KUKA KRL program: XmlDualMove_better.src

&ACCESS RV
&REL 1
&PARAM DISKPATH = KRC:\R1\Program
&PARAM SensorITMASK = *
&PARAM TEMPLATE = C:\KRC\Roboter\Template\vorgabe
DEF XmlDualMove_better( )

; ============================================================================
; XmlDualMove_better - robot-interpreter side of the ROS2 link, BATCH capable
; ============================================================================
; RELATIONSHIP WITH XmlDualMove.src
;   XmlDualMove.src        baseline used for the KRL vs MoveIt2 comparative
;                          study.  Untouched.  Still selectable and still
;                          works against XmlDualMove_better.xml, because that
;                          channel config is a strict superset.
;   XmlDualMove_better.src this file: everything the baseline does, PLUS the
;                          batch mode.  Only ONE of the two is selected at a
;                          time; they never run together.
;
; WHAT BATCH MODE CHANGES
;   The baseline executes one point per network round trip: ROS sends a point,
;   waits for the robot to arrive, then sends the next.  Over 100+ trajectory
;   points that dead time is what produces the advance-brake-advance pattern.
;
;   In batch mode ROS ships a block of up to XD_BATCH_MAX points, the SPS drops
;   the whole block into the mailbox in one go, and this program walks it
;   locally with no network in the inner loop.
;
;   Every point is STILL an exact-stop PTP.  No C_PTP, no blending, no SLIN,
;   no Cartesian.  The motion type is identical; only the waiting changes.
;
; ADVANCE RUN
;   KRL executes assignments during the advance run, and $ADVANCE defaults to
;   3 (KSS 8.2 System Integrators, 7.5.3 "Advance run", p. 208: default 3,
;   maximum 5).  Left alone, XD_BATCH_CONSUMED_COUNT would run up to $ADVANCE
;   points ahead of the real motion and the abort check would read stale state.
;
;   This program does NOT write $ADVANCE.  It forces the advance-run stop once
;   per point with WAIT SEC 0 instead, which is the documented way to make an
;   instruction run in the main run, and which costs nothing here because every
;   point is already an exact stop.  $ADVANCE = 0 would be legal (0 is inside
;   the documented range) but it also makes approximate positioning impossible,
;   and blending is where this design is headed next.
;
;   The WAIT SEC 0.1 of the main loop is NOT touched: same place, same value.
;   It simply does not sit between the points of one batch.
; ============================================================================
; THIS PROGRAM CONTAINS NO EthernetKRL CALLS.
;
; SPS.SUB owns the EKI channel: it opens it, drains the receive buffer on
; every cycle and publishes the last valid command into the XD_ mailbox in
; $CONFIG.DAT.  This program only reads that mailbox.  Consequences:
;
;   * Telemetry no longer depends on this program running.  DEMO26 or any
;     other KRL program can be selected and Ubuntu keeps receiving data.
;   * The receive buffer is never blocked by the robot interpreter, which is
;     what used to fill the EKI memory and raise EKI01280.
;   * The manual warns against reading one channel from both interpreters
;     (EKI_Get empties the memory), so all reading stays in the SPS.
;
; SAFETY MODEL
;   * On start-up the current mailbox Seq is taken as a BASELINE and is never
;     executed.  A command that arrived while DEMO26 was running can never
;     move the robot just because this program was selected afterwards.
;   * A Seq is marked handled BEFORE acting on it, so a given Seq can move
;     the robot or drive the gripper at most once.  The Ubuntu heartbeat
;     deliberately repeats the same Seq and is therefore inert.
;   * Gripper and motion are independent: EnableMove=FALSE with
;     GripperCommand 0 or 1 performs a gripper-only action.
;
; ORDER OF EXECUTION for a new Seq:  validate -> gripper -> motion.
; ============================================================================

;FOLD Declaration
  INT i
  INT cmdSeq
  INT cmdSeqCheck
  INT handledSeq
  INT gripperCmd

  DECL AXIS axisTarget
  DECL E6POS cartesianTarget

  BOOL snapshotOK
  BOOL isAxisMode
  BOOL isCartesianMode

  BOOL enableMove
  BOOL limitsOK
  BOOL readyToMove
  BOOL moveExecuted
  BOOL deltaOK
  BOOL velocityOK
  BOOL hasTrajectoryVelocity

  REAL targetA1
  REAL targetA2
  REAL targetA3
  REAL targetA4
  REAL targetA5
  REAL targetA6

  REAL targetX
  REAL targetY
  REAL targetZ
  REAL targetA
  REAL targetB
  REAL targetC
  REAL ptpVelocityPct

  REAL errorA1
  REAL errorA2
  REAL errorA3
  REAL errorA4
  REAL errorA5
  REAL errorA6

  REAL errorX
  REAL errorY
  REAL errorZ
  REAL errorA
  REAL errorB
  REAL errorC

  REAL MAX_DELTA_JOINT
  REAL MAX_DELTA_POS
  REAL MAX_DELTA_ORI

  ; ---- BATCH MODE ----
  INT batchSeq
  INT batchSeqCheck
  INT handledBatchSeq
  INT batchCount
  INT batchI
  INT savedAdvance
  REAL batchVelPct
  REAL batchErr
  BOOL batchSnapshotOK
  BOOL batchRunning
  BOOL batchPointOK
  BOOL hasBatchVelocity
  BOOL batchLoaded
  BOOL batchGateOK
  BOOL batchVelocityOK
  ; Ultimo punto ENTREGADO al planificador.  La validacion de salto se hace
  ; contra este valor y NO contra $AXIS_ACT: con aproximacion activa el robot
  ; va por detras del interprete a proposito, asi que $AXIS_ACT no dice donde
  ; estara cuando se ejecute el punto que se esta validando.  Ademas leer
  ; $AXIS_ACT dentro del encadenado obligaria a una parada del avance, que es
  ; justo lo que impide aproximar (KSS 8.2 SI, 8.5, p. 224).
  REAL prevA1
  REAL prevA2
  REAL prevA3
  REAL prevA4
  REAL prevA5
  REAL prevA6
  INT localBatchSeq
  INT localBatchCount
  REAL localBatchVelPct
  DECL AXIS batchTarget

  ; LOCAL copy of the batch.  The mailbox holds ONE batch slot, so executing
  ; straight out of it would mean ROS could not load the next batch until the
  ; current one finished - the very network gap batch mode exists to remove.
  ; Copying to locals frees the mailbox the moment execution starts, so ROS
  ; can refill it while the robot is still moving.
  REAL localA1[20]
  REAL localA2[20]
  REAL localA3[20]
  REAL localA4[20]
  REAL localA5[20]
  REAL localA6[20]
;ENDFOLD (Declaration)

;FOLD INI
  ;FOLD BASISTECH INI
    BAS (#INITMOV,0 )
  ;ENDFOLD (BASISTECH INI)

  ;FOLD USER INI
    ;Reads targets from the XD_ mailbox published by SPS.SUB.
    ;Supports BOTH Axis (A1-A6) and Cartesian (X,Y,Z,A,B,C) modes.
    ;Movement must be enabled by the responsible operator via the bridge.
  ;ENDFOLD (USER INI)
;ENDFOLD (INI)

;FOLD Initialize data
  cmdSeq = 0
  cmdSeqCheck = 0
  gripperCmd = -1

  snapshotOK = FALSE
  enableMove = FALSE
  limitsOK = FALSE
  readyToMove = FALSE
  moveExecuted = FALSE
  deltaOK = FALSE
  velocityOK = FALSE
  hasTrajectoryVelocity = FALSE
  isAxisMode = FALSE
  isCartesianMode = FALSE

  targetA1 = $AXIS_ACT.A1
  targetA2 = $AXIS_ACT.A2
  targetA3 = $AXIS_ACT.A3
  targetA4 = $AXIS_ACT.A4
  targetA5 = $AXIS_ACT.A5
  targetA6 = $AXIS_ACT.A6

  targetX = $POS_ACT.X
  targetY = $POS_ACT.Y
  targetZ = $POS_ACT.Z
  targetA = $POS_ACT.A
  targetB = $POS_ACT.B
  targetC = $POS_ACT.C
  ptpVelocityPct = 0.0

  errorA1 = 0.0
  errorA2 = 0.0
  errorA3 = 0.0
  errorA4 = 0.0
  errorA5 = 0.0
  errorA6 = 0.0

  errorX = 0.0
  errorY = 0.0
  errorZ = 0.0
  errorA = 0.0
  errorB = 0.0
  errorC = 0.0

  MAX_DELTA_JOINT = 10.0
  MAX_DELTA_POS = 100.0  ; 100 mm jump max in X, Y, Z
  MAX_DELTA_ORI = 20.0   ; 20 degrees jump max in A, B, C

  axisTarget = $AXIS_ACT
  cartesianTarget = $POS_ACT

  ; ---- BASELINE ----
  ; Whatever is sitting in the mailbox right now belongs to the past: it may
  ; have arrived while DEMO26 was running, or be the last command of an
  ; earlier ROS2 session.  Treating it as already handled is what stops this
  ; program from moving the moment it is selected.
  handledSeq = XD_CMD_SEQ

  ; Same baseline rule for the batch: whatever batch is sitting in the mailbox
  ; when this program is selected belongs to the past and is never executed.
  handledBatchSeq = XD_BATCH_SEQ

  batchSeq = 0
  batchSeqCheck = 0
  batchCount = 0
  batchI = 0
  savedAdvance = 3
  batchVelPct = 0.0
  batchErr = 0.0
  batchSnapshotOK = FALSE
  batchRunning = FALSE
  batchPointOK = FALSE
  hasBatchVelocity = FALSE
  batchLoaded = FALSE
  batchGateOK = FALSE
  batchVelocityOK = FALSE
  prevA1 = 0.0
  prevA2 = 0.0
  prevA3 = 0.0
  prevA4 = 0.0
  prevA5 = 0.0
  prevA6 = 0.0
  localBatchSeq = 0
  localBatchCount = 0
  localBatchVelPct = 0.0
  batchTarget = $AXIS_ACT

  XD_BATCH_ACTIVE = FALSE
  XD_BATCH_CONSUMED_COUNT = 0

  XD_MOVE_READY = FALSE
  XD_LIMITS_OK = FALSE
  XD_DELTA_OK = FALSE
;ENDFOLD (Initialize data)

;FOLD Configure motion parameters
  $BWDSTART = FALSE

  ; Default TOOL and BASE (modify if your setup requires specific ones)
  $TOOL = $NULLFRAME
  $BASE = $NULLFRAME
;ENDFOLD (Configure motion parameters)

;FOLD Move command loop
LOOP

  ;FOLD Snapshot the mailbox
    ; Seqlock read: XD_CMD_SEQ is written LAST by the SPS, so reading it
    ; before and after the payload detects a publish that landed mid-copy.
    ; A torn snapshot is simply discarded and retried next cycle.
    snapshotOK = FALSE

    IF XD_CMD_UPDATING == FALSE THEN
      cmdSeqCheck = XD_CMD_SEQ

      targetA1 = XD_TARGET_A1
      targetA2 = XD_TARGET_A2
      targetA3 = XD_TARGET_A3
      targetA4 = XD_TARGET_A4
      targetA5 = XD_TARGET_A5
      targetA6 = XD_TARGET_A6

      targetX = XD_TARGET_X
      targetY = XD_TARGET_Y
      targetZ = XD_TARGET_Z
      targetA = XD_TARGET_A
      targetB = XD_TARGET_B
      targetC = XD_TARGET_C

      enableMove = XD_ENABLE_MOVE
      gripperCmd = XD_GRIPPER_COMMAND
      ptpVelocityPct = XD_TRAJ_PTP_VEL_PCT
      isAxisMode = XD_AXIS_MODE
      isCartesianMode = XD_CART_MODE

      IF (XD_CMD_UPDATING == FALSE) AND (XD_CMD_SEQ == cmdSeqCheck) THEN
        cmdSeq = cmdSeqCheck
        snapshotOK = TRUE
      ENDIF
    ENDIF
  ;ENDFOLD (Snapshot the mailbox)

  ;FOLD Snapshot the batch mailbox
    ; Same seqlock idea as the single-point snapshot: XD_BATCH_SEQ is written
    ; LAST by the SPS, so reading it before and after the payload detects a
    ; publish that landed mid-copy.  A torn batch is discarded and retried.
    batchSnapshotOK = FALSE

    IF XD_CMD_UPDATING == FALSE THEN
      batchSeqCheck = XD_BATCH_SEQ
      batchCount = XD_BATCH_COUNT
      batchVelPct = XD_BATCH_PTP_VEL_PCT

      IF (XD_CMD_UPDATING == FALSE) AND (XD_BATCH_SEQ == batchSeqCheck) THEN
        batchSeq = batchSeqCheck
        batchSnapshotOK = TRUE
      ENDIF
    ENDIF

    ; A batch mailbox reset follows the same rule as the single-point one.
    IF batchSnapshotOK == TRUE THEN
      IF batchSeq == 0 THEN
        handledBatchSeq = 0
      ENDIF
    ENDIF

    ; Velocity validation, identical rule to the single-point path.
    hasBatchVelocity = FALSE
    IF (batchVelPct > 0.0) AND (batchVelPct <= 100.0) THEN
      hasBatchVelocity = TRUE
    ENDIF
  ;ENDFOLD (Snapshot the batch mailbox)

  ;FOLD Follow a mailbox reset
    ; XD_CMD_SEQ == 0 is the sentinel the SPS writes when it (re)opens the
    ; channel: the mailbox holds no command at all.  There is nothing from
    ; the past to protect against, so the handled marker follows it down.
    ; Without this, a fresh ROS2 session that restarts its counter at 1 could
    ; have its very first command silently ignored.
    IF snapshotOK == TRUE THEN
      IF cmdSeq == 0 THEN
        handledSeq = 0
      ENDIF
    ENDIF
  ;ENDFOLD (Follow a mailbox reset)

  ;FOLD Calculate error target - actual
    IF isAxisMode THEN
      errorA1 = targetA1 - $AXIS_ACT.A1
      errorA2 = targetA2 - $AXIS_ACT.A2
      errorA3 = targetA3 - $AXIS_ACT.A3
      errorA4 = targetA4 - $AXIS_ACT.A4
      errorA5 = targetA5 - $AXIS_ACT.A5
      errorA6 = targetA6 - $AXIS_ACT.A6
    ENDIF

    IF isCartesianMode THEN
      errorX = targetX - $POS_ACT.X
      errorY = targetY - $POS_ACT.Y
      errorZ = targetZ - $POS_ACT.Z
      errorA = targetA - $POS_ACT.A
      errorB = targetB - $POS_ACT.B
      errorC = targetC - $POS_ACT.C
    ENDIF
  ;ENDFOLD (Calculate error target - actual)

  ;FOLD Validate limits
    limitsOK = TRUE

    IF isAxisMode THEN
      IF targetA1 < -160.0 THEN
        limitsOK = FALSE
      ENDIF
      IF targetA1 > 160.0 THEN
        limitsOK = FALSE
      ENDIF
      IF targetA2 < -180.0 THEN
        limitsOK = FALSE
      ENDIF
      IF targetA2 > 35.0 THEN
        limitsOK = FALSE
      ENDIF
      IF targetA3 < -110.0 THEN
        limitsOK = FALSE
      ENDIF
      IF targetA3 > 146.0 THEN
        limitsOK = FALSE
      ENDIF
      IF targetA4 < -175.0 THEN
        limitsOK = FALSE
      ENDIF
      IF targetA4 > 175.0 THEN
        limitsOK = FALSE
      ENDIF
      IF targetA5 < -110.0 THEN
        limitsOK = FALSE
      ENDIF
      IF targetA5 > 110.0 THEN
        limitsOK = FALSE
      ENDIF
      IF targetA6 < -340.0 THEN
        limitsOK = FALSE
      ENDIF
      IF targetA6 > 340.0 THEN
        limitsOK = FALSE
      ENDIF
    ENDIF

    ; Note: Cartesian limits are harder to define safely without a known workspace.
    ; Native KUKA reachability will prevent unsafe poses, but you can add boundary boxes here if needed.
  ;ENDFOLD (Validate limits)

  XD_LIMITS_OK = limitsOK

  ;FOLD Validate delta (max jump per command)
    deltaOK = TRUE

    IF isAxisMode THEN
      IF (errorA1 > MAX_DELTA_JOINT) OR (errorA1 < -MAX_DELTA_JOINT) THEN
        deltaOK = FALSE
      ENDIF
      IF (errorA2 > MAX_DELTA_JOINT) OR (errorA2 < -MAX_DELTA_JOINT) THEN
        deltaOK = FALSE
      ENDIF
      IF (errorA3 > MAX_DELTA_JOINT) OR (errorA3 < -MAX_DELTA_JOINT) THEN
        deltaOK = FALSE
      ENDIF
      IF (errorA4 > MAX_DELTA_JOINT) OR (errorA4 < -MAX_DELTA_JOINT) THEN
        deltaOK = FALSE
      ENDIF
      IF (errorA5 > MAX_DELTA_JOINT) OR (errorA5 < -MAX_DELTA_JOINT) THEN
        deltaOK = FALSE
      ENDIF
      IF (errorA6 > MAX_DELTA_JOINT) OR (errorA6 < -MAX_DELTA_JOINT) THEN
        deltaOK = FALSE
      ENDIF
    ENDIF

    IF isCartesianMode THEN
      IF (errorX > MAX_DELTA_POS) OR (errorX < -MAX_DELTA_POS) THEN
        deltaOK = FALSE
      ENDIF
      IF (errorY > MAX_DELTA_POS) OR (errorY < -MAX_DELTA_POS) THEN
        deltaOK = FALSE
      ENDIF
      IF (errorZ > MAX_DELTA_POS) OR (errorZ < -MAX_DELTA_POS) THEN
        deltaOK = FALSE
      ENDIF
      IF (errorA > MAX_DELTA_ORI) OR (errorA < -MAX_DELTA_ORI) THEN
        deltaOK = FALSE
      ENDIF
      IF (errorB > MAX_DELTA_ORI) OR (errorB < -MAX_DELTA_ORI) THEN
        deltaOK = FALSE
      ENDIF
      IF (errorC > MAX_DELTA_ORI) OR (errorC < -MAX_DELTA_ORI) THEN
        deltaOK = FALSE
      ENDIF
    ENDIF
  ;ENDFOLD (Validate delta)

  XD_DELTA_OK = deltaOK

  ;FOLD Validate trajectory PTP velocity
    ; 0.0 identifies SEND manual/legacy and leaves the current programmed PTP
    ; velocity untouched. Positive values belong only to AxisTarget trajectory
    ; commands. Invalid mailbox values block motion.
    velocityOK = FALSE
    hasTrajectoryVelocity = FALSE

    IF ptpVelocityPct == 0.0 THEN
      velocityOK = TRUE
    ENDIF
    IF (ptpVelocityPct > 0.0) AND (ptpVelocityPct <= 100.0) THEN
      velocityOK = TRUE
      hasTrajectoryVelocity = TRUE
    ENDIF
    IF isCartesianMode AND hasTrajectoryVelocity THEN
      velocityOK = FALSE
    ENDIF
  ;ENDFOLD (Validate trajectory PTP velocity)

  ;FOLD Build target from mailbox
    IF isAxisMode THEN
      axisTarget = $AXIS_ACT
      axisTarget.A1 = targetA1
      axisTarget.A2 = targetA2
      axisTarget.A3 = targetA3
      axisTarget.A4 = targetA4
      axisTarget.A5 = targetA5
      axisTarget.A6 = targetA6
    ENDIF

    IF isCartesianMode THEN
      cartesianTarget = $POS_ACT
      cartesianTarget.X = targetX
      cartesianTarget.Y = targetY
      cartesianTarget.Z = targetZ
      cartesianTarget.A = targetA
      cartesianTarget.B = targetB
      cartesianTarget.C = targetC
    ENDIF
  ;ENDFOLD (Build target from mailbox)

  ;FOLD Determine readyToMove
    readyToMove = FALSE

    IF enableMove == TRUE THEN
      IF limitsOK == TRUE THEN
        IF deltaOK == TRUE THEN
          IF velocityOK == TRUE THEN
            IF snapshotOK == TRUE THEN
              readyToMove = TRUE
            ENDIF
          ENDIF
        ENDIF
      ENDIF
    ENDIF

    IF XD_EKI_ACTIVE == FALSE THEN
      readyToMove = FALSE
    ENDIF
    IF (isAxisMode == FALSE) AND (isCartesianMode == FALSE) THEN
      readyToMove = FALSE
    ENDIF

    XD_MOVE_READY = readyToMove
  ;ENDFOLD (Determine readyToMove)

  ;FOLD Act on a NEW sequence only
    ; A Seq is acted on exactly once.  handledSeq is advanced BEFORE the
    ; action, so nothing can replay it: not the heartbeat, not a restart.
    ;
    ; BATCH GUARD: a batch packet also carries Command/Seq, so without this
    ; guard the single-point block would fire on the batch packet and drive
    ; the robot to XD_TARGET_A1..A6 before the batch even starts.  While a
    ; batch is pending or running, the single-point path stands down.
    ; Ordinary single-point commands are unaffected: with no batch in the
    ; mailbox, batchSeq equals handledBatchSeq and this guard is transparent.
    IF (batchSeq == handledBatchSeq) AND (batchRunning == FALSE) THEN
    IF snapshotOK == TRUE THEN
      IF cmdSeq > 0 THEN
        IF cmdSeq <> handledSeq THEN
          IF XD_EKI_ACTIVE == TRUE THEN

            handledSeq = cmdSeq

            ;FOLD Gripper action
              ; -1 = do nothing (the bridge default), 0 = open, 1 = close.
              ; The SPS has already rejected any other value.
              IF gripperCmd == 0 THEN
                GRPg_SetStateAndCheck(1, 1, 0.2, 1)
              ENDIF
              IF gripperCmd == 1 THEN
                GRPg_SetStateAndCheck(1, 2, 0.2, 1)
              ENDIF
            ;ENDFOLD (Gripper action)

            ;FOLD Motion
              IF readyToMove == TRUE THEN
                IF isAxisMode THEN
                  IF hasTrajectoryVelocity THEN
                    BAS (#VEL_PTP,ptpVelocityPct)
                  ENDIF
                  PTP axisTarget
                ENDIF

                IF isCartesianMode THEN
                  PTP cartesianTarget
                ENDIF

                moveExecuted = TRUE
                XD_LAST_MOVE_SEQ = cmdSeq
                XD_MOVE_EXECUTED = TRUE
              ENDIF
            ;ENDFOLD (Motion)

          ENDIF
        ENDIF
      ENDIF
    ENDIF
    ENDIF
  ;ENDFOLD (Act on a NEW sequence only)

  ;FOLD Execute a NEW batch
    ; A batch is acted on exactly once, same contract as a single Seq:
    ; handledBatchSeq advances BEFORE the first point, so nothing can replay
    ; it after a restart or a repeated packet.
    ;
    ; REFILL WHILE MOVING
    ;   The mailbox has ONE batch slot.  Executing straight out of it would
    ;   force ROS to wait for the batch to finish before loading the next,
    ;   reintroducing one network gap per batch.  So the batch is copied into
    ;   local arrays first: the mailbox is free again immediately and ROS can
    ;   refill it while the robot is still moving through the local copy.
    ;   The WHILE below then picks up that next batch with no gap at all.
    ;
    ;   If no new batch has arrived by the time the local copy runs out, the
    ;   WHILE exits and the outer loop simply waits - same behaviour as the
    ;   baseline when no command is present.
    ; Entry gate for a new batch.  These five conditions were five nested
    ; IFs.  KRL allows at most 10 nested control structures and that pushed
    ; the batch loop to depth 12, so the controller rejected the file with
    ; error 2218.  Same conditions, same order, same outcome - the only
    ; thing that changed is the nesting depth.  Do NOT re-nest them.
    batchGateOK = (batchSnapshotOK == TRUE) AND (batchSeq > 0)
    batchGateOK = batchGateOK AND (batchSeq <> handledBatchSeq)
    batchGateOK = batchGateOK AND (XD_EKI_ACTIVE == TRUE)
    batchGateOK = batchGateOK AND (XD_ENABLE_MOVE == TRUE)
    IF batchGateOK == TRUE THEN

      ; EL LOTE CONSUME TAMBIEN Command/Seq.
      ; Un paquete de lote lleva ADEMAS Command/Seq y Command/AxisTarget.
      ; Ese AxisTarget es relleno inerte: la posicion que tenia el robot
      ; cuando ROS envio el lote.  Pero el bloque de punto suelto no sabe
      ; que es relleno.  Al terminar el lote su puerta se reabre
      ; (batchSeq == handledBatchSeq, batchRunning == FALSE), encuentra un
      ; Seq que nadie ha atendido y lo ejecuta como un PTP normal: el robot
      ; vuelve al punto donde EMPEZO el lote.
      ; En los tramos largos la validacion de delta lo frena (recorridos de
      ; 30-90 grados contra MAX_DELTA_JOINT = 10.0).  En los tramos cortos
      ; de aproximacion y retirada NO: P3->P4 son 9.888 grados, y P4->P5
      ; otros 9.710.  Medido: el robot bajaba, agarraba, subia, volvia a
      ; bajar y a subir varias veces antes de seguir - un rebote por cada
      ; tramo corto.
      ; Atender el Seq aqui es correcto por definicion: el paquete YA se ha
      ; consumido, por el camino de lote.  Nada se pierde, porque el
      ; AxisTarget de un paquete de lote nunca fue un destino real y su
      ; GripperCommand es siempre -1.
      handledSeq = cmdSeq

      ; A stale abort from a previous batch must not kill this one.
      XD_ABORT_BATCH = FALSE
      XD_BATCH_ACTIVE = TRUE
      batchRunning = TRUE

      ; Every point inside the batch forces its own advance-run stop
      ; with WAIT SEC 0 (see the FOR below).  $ADVANCE is deliberately
      ; NOT written here.  It was once suspected of raising KSS01422;
      ; that was never proven - the error kept firing after every write
      ; to $ADVANCE had been removed - so that claim is withdrawn.
      ; WAIT SEC 0 stays because it is the documented mechanism, not
      ; because $ADVANCE is dangerous.

      ; Ancla de la cadena de validacion.  Esta es la UNICA lectura de
      ; $AXIS_ACT de todo el camino de movimiento, y esta antes del primer
      ; PTP, donde una parada del avance no cuesta nada.  A partir de aqui
      ; cada punto se valida contra el ANTERIOR, que es exactamente lo que
      ; preflight() de ROS ya comprueba sobre el archivo entero.
      WAIT SEC 0
      prevA1 = $AXIS_ACT.A1
      prevA2 = $AXIS_ACT.A2
      prevA3 = $AXIS_ACT.A3
      prevA4 = $AXIS_ACT.A4
      prevA5 = $AXIS_ACT.A5
      prevA6 = $AXIS_ACT.A6

      WHILE batchRunning == TRUE

        ;FOLD Copy the mailbox batch into the local arrays
          ; Seqlock read, same idea as the single-point snapshot.
          batchLoaded = FALSE

          IF XD_CMD_UPDATING == FALSE THEN
            batchSeqCheck = XD_BATCH_SEQ
            localBatchCount = XD_BATCH_COUNT
            localBatchVelPct = XD_BATCH_PTP_VEL_PCT

            IF localBatchCount > 0 THEN
              IF localBatchCount <= XD_BATCH_MAX THEN
                FOR batchI = 1 TO localBatchCount
                  localA1[batchI] = XD_BATCH_A1[batchI]
                  localA2[batchI] = XD_BATCH_A2[batchI]
                  localA3[batchI] = XD_BATCH_A3[batchI]
                  localA4[batchI] = XD_BATCH_A4[batchI]
                  localA5[batchI] = XD_BATCH_A5[batchI]
                  localA6[batchI] = XD_BATCH_A6[batchI]
                ENDFOR

                IF (XD_CMD_UPDATING == FALSE) AND (XD_BATCH_SEQ == batchSeqCheck) THEN
                  IF batchSeqCheck <> handledBatchSeq THEN
                    localBatchSeq = batchSeqCheck
                    batchLoaded = TRUE
                  ENDIF
                ENDIF
              ENDIF
            ENDIF
          ENDIF

          ; Nothing new in the mailbox: leave the batch loop and let
          ; the outer loop wait.  The robot does not move.
          IF batchLoaded == FALSE THEN
            batchRunning = FALSE
          ENDIF
        ;ENDFOLD (Copy the mailbox batch)

        IF batchRunning == TRUE THEN

          ; Claimed BEFORE the first point: nothing can replay it.
          handledBatchSeq = localBatchSeq

          ; XD_BATCH_CONSUMED_COUNT is NOT reset here any more.  It used to
          ; restart at 0 on every batch, which forced ROS to reconstruct the
          ; segment total as "points of the finished batches + this one" -
          ; and ROS has no way to know which batch is executing, only which
          ; one it last SENT.  The moment it pre-loaded the next batch its
          ; total jumped a whole batch ahead of reality, the segment was
          ; declared finished before the last batch ran, and the robot never
          ; reached the end point.
          ; It is now a free-running total of batch points executed since the
          ; channel opened.  ROS takes a baseline at the start of each segment
          ; and subtracts.  A missed telemetry sample can no longer lose a
          ; reset, because there are no resets left to miss.

          ; Velocity gate, now the SAME rule as the single-point path.
          ; The SPS publishes -1.0 into XD_BATCH_PTP_VEL_PCT whenever the
          ; value on the wire fell outside (0, 100].  The single-point
          ; path turns that into velocityOK = FALSE and refuses to move.
          ; This path only used the value to decide whether to CALL BAS,
          ; so a rejected velocity silently ran the whole batch at
          ; whatever PTP velocity happened to be programmed.  Now:
          ;   0.0        keep the currently programmed velocity
          ;   (0, 100]   program it with BAS(#VEL_PTP, ...)
          ;   anything else -> the batch stops before the first point.
          ; Clearing batchRunning here is enough: every iteration of the
          ; FOR below only moves inside IF batchRunning == TRUE.
          batchVelocityOK = FALSE
          hasBatchVelocity = FALSE
          IF localBatchVelPct == 0.0 THEN
            batchVelocityOK = TRUE
          ENDIF
          IF (localBatchVelPct > 0.0) AND (localBatchVelPct <= 100.0) THEN
            batchVelocityOK = TRUE
            hasBatchVelocity = TRUE
          ENDIF
          IF batchVelocityOK == FALSE THEN
            batchRunning = FALSE
          ENDIF
          IF hasBatchVelocity THEN
            BAS (#VEL_PTP,localBatchVelPct)
          ENDIF

          FOR batchI = 1 TO localBatchCount

            ; NO hay parada del avance aqui.  La habia (WAIT SEC 0) y era
            ; precisamente lo que impedia encadenar los puntos: KSS 8.2 SI,
            ; 8.5, p. 224 - "Approximate positioning is not possible if the
            ; motion instruction is followed by an instruction that triggers
            ; an advance run stop".  Sin ella el interprete planifica por
            ; delante y los PTP se solapan, que es todo el objetivo.
            ;
            ; Consecuencia asumida: estas puertas se evaluan en el AVANCE,
            ; hasta $ADVANCE puntos por delante del movimiento real.  Un
            ; abort no frena en el punto siguiente sino tras los bloques ya
            ; planificados - que es como XD_ABORT_BATCH estuvo documentado
            ; desde el principio ("termina el PTP en vuelo").

            ;FOLD Local gates - re-checked before EVERY point
              ; All local: no network, so this adds no latency back.
              IF XD_ABORT_BATCH == TRUE THEN
                batchRunning = FALSE
              ENDIF
              IF XD_ENABLE_MOVE == FALSE THEN
                batchRunning = FALSE
              ENDIF
              IF XD_EKI_ACTIVE == FALSE THEN
                batchRunning = FALSE
              ENDIF
            ;ENDFOLD (Local gates)

            IF batchRunning == TRUE THEN

              ;FOLD Build this point from the LOCAL copy
                ; batchTarget es DECL AXIS: A1..A6 y nada mas, y los seis se
                ; asignan aqui.  El "batchTarget = $AXIS_ACT" que habia como
                ; semilla era redundante y metia una lectura de la posicion
                ; real en mitad del encadenado.
                batchTarget.A1 = localA1[batchI]
                batchTarget.A2 = localA2[batchI]
                batchTarget.A3 = localA3[batchI]
                batchTarget.A4 = localA4[batchI]
                batchTarget.A5 = localA5[batchI]
                batchTarget.A6 = localA6[batchI]
              ;ENDFOLD (Build this point)

              ;FOLD Validate this point - same limits as the baseline
                batchPointOK = TRUE

                ; MISMOS limites y misma consecuencia que antes: lo unico
                ; que cambia es que cada eje se comprueba con UNA sentencia
                ; en vez de dos, igual que ya se hacia justo debajo con el
                ; delta.  Son 18 lineas menos de interprete POR PUNTO.
                ; KSS 8.2 SI, 7.5.3, p. 208: el avance planifica hasta
                ; $ADVANCE bloques, pero "the actual number is dependent on
                ; the capacity of the computer".  Cuanto menos cuesta cada
                ; punto, mas lejos llega el avance con el mismo $ADVANCE, y
                ; menos probable es que la cola de movimiento se vacie entre
                ; dos PTP encadenados.  Ninguna proteccion se toca.
                IF (batchTarget.A1 < -160.0) OR (batchTarget.A1 > 160.0) THEN
                  batchPointOK = FALSE
                ENDIF
                IF (batchTarget.A2 < -180.0) OR (batchTarget.A2 > 35.0) THEN
                  batchPointOK = FALSE
                ENDIF
                IF (batchTarget.A3 < -110.0) OR (batchTarget.A3 > 146.0) THEN
                  batchPointOK = FALSE
                ENDIF
                IF (batchTarget.A4 < -175.0) OR (batchTarget.A4 > 175.0) THEN
                  batchPointOK = FALSE
                ENDIF
                IF (batchTarget.A5 < -110.0) OR (batchTarget.A5 > 110.0) THEN
                  batchPointOK = FALSE
                ENDIF
                IF (batchTarget.A6 < -340.0) OR (batchTarget.A6 > 340.0) THEN
                  batchPointOK = FALSE
                ENDIF
              ;ENDFOLD (Validate this point)

              ;FOLD Validate delta against the PREVIOUS point
                ; Mismo umbral MAX_DELTA_JOINT y misma consecuencia que
                ; antes; lo que cambia es la referencia.  Con aproximacion
                ; activa el robot va por detras del interprete a proposito,
                ; asi que $AXIS_ACT no dice donde estara el robot cuando
                ; ejecute ESTE punto - comparar contra el seria comparar
                ; contra el pasado.  prevA1..A6 es el punto anterior de la
                ; cadena, anclado en la posicion REAL antes del primer PTP.
                ; Es la misma comprobacion que preflight() de ROS aplica al
                ; archivo entero antes de enviar nada.
                batchErr = batchTarget.A1 - prevA1
                IF (batchErr > MAX_DELTA_JOINT) OR (batchErr < -MAX_DELTA_JOINT) THEN
                  batchPointOK = FALSE
                ENDIF
                batchErr = batchTarget.A2 - prevA2
                IF (batchErr > MAX_DELTA_JOINT) OR (batchErr < -MAX_DELTA_JOINT) THEN
                  batchPointOK = FALSE
                ENDIF
                batchErr = batchTarget.A3 - prevA3
                IF (batchErr > MAX_DELTA_JOINT) OR (batchErr < -MAX_DELTA_JOINT) THEN
                  batchPointOK = FALSE
                ENDIF
                batchErr = batchTarget.A4 - prevA4
                IF (batchErr > MAX_DELTA_JOINT) OR (batchErr < -MAX_DELTA_JOINT) THEN
                  batchPointOK = FALSE
                ENDIF
                batchErr = batchTarget.A5 - prevA5
                IF (batchErr > MAX_DELTA_JOINT) OR (batchErr < -MAX_DELTA_JOINT) THEN
                  batchPointOK = FALSE
                ENDIF
                batchErr = batchTarget.A6 - prevA6
                IF (batchErr > MAX_DELTA_JOINT) OR (batchErr < -MAX_DELTA_JOINT) THEN
                  batchPointOK = FALSE
                ENDIF
              ;ENDFOLD (Validate delta)

              ;FOLD Move
                IF batchPointOK == TRUE THEN
                  ; C_PTP = aproximacion PTP-PTP.  KSS 8.2 SI, 10.5.1,
                  ; p. 297: "The specification C_PTP is sufficient for
                  ; PTP-PTP approximate positioning".  La distancia de
                  ; aproximacion sale de los valores por defecto que deja
                  ; BAS(#INITMOV,0) al principio del programa; aqui no se
                  ; escribe $APO para no meter otra escritura a una
                  ; variable de sistema en el camino critico.
                  ;
                  ; En el ULTIMO punto de la secuencia no hay bloque de
                  ; movimiento siguiente en el avance, asi que el
                  ; controlador no puede aproximar y para exacto por si
                  ; solo (KSS 8.2 SI, 8.5, p. 225).  Esa es la parada en
                  ; el punto final del segmento, y sale gratis.
                  PTP batchTarget C_PTP
                  ; Contador de progreso.  AQUI HABIA UN TRIGGER y era un
                  ; error: "TRIGGER ... DO XD_BATCH_CONSUMED_COUNT =
                  ; XD_BATCH_CONSUMED_COUNT + 1" es una lectura-modificacion-
                  ; escritura de la MISMA global, y con el avance activo hay
                  ; hasta $ADVANCE disparadores registrados a la vez que leen
                  ; todos el mismo valor de partida.  Resultado medido: 20
                  ; puntos ejecutados, el contador marcaba 4.  ROS no llegaba
                  ; nunca al umbral de reposicion y no mandaba el lote 2.
                  ;
                  ; Ahora es una asignacion normal, que se ejecuta en el
                  ; AVANCE: cuenta puntos PLANIFICADOS, no alcanzados, y va
                  ; por delante del robot como mucho $ADVANCE puntos (maximo
                  ; 5 segun KSS 8.2 SI, 7.5.3, p. 208).  Adelantarse es
                  ; inofensivo para reponer lotes - de hecho conviene -, y la
                  ; llegada REAL al punto final del segmento la comprueba ROS
                  ; contra AxisActual, que no depende de este contador.
                  XD_BATCH_CONSUMED_COUNT = XD_BATCH_CONSUMED_COUNT + 1
                  XD_LAST_MOVE_SEQ = localBatchSeq
                  XD_MOVE_EXECUTED = TRUE
                  ; La cadena avanza: el punto que se acaba de entregar
                  ; pasa a ser la referencia del siguiente.
                  prevA1 = batchTarget.A1
                  prevA2 = batchTarget.A2
                  prevA3 = batchTarget.A3
                  prevA4 = batchTarget.A4
                  prevA5 = batchTarget.A5
                  prevA6 = batchTarget.A6
                ELSE
                  ; A point that fails its own validation stops the
                  ; batch.  Skipping it silently would move the robot
                  ; along a path nobody validated.
                  batchRunning = FALSE
                ENDIF
              ;ENDFOLD (Move)

            ENDIF
          ENDFOR

        ENDIF
      ENDWHILE

      ; Release the batch.
      batchRunning = FALSE
      XD_BATCH_ACTIVE = FALSE
      XD_ABORT_BATCH = FALSE

    ENDIF
  ;ENDFOLD (Execute a NEW batch)

  WAIT SEC 0.1

ENDLOOP
;ENDFOLD (Move command loop)

; No EKI_Close here: the channel belongs to SPS.SUB and must survive this
; program being deselected.  That is the whole point of the redesign.

END
